FUNCTION_BLOCK FB_VirtualControlBox IMPLEMENTS I_ControlBox
VAR_INPUT
END_VAR
VAR_OUTPUT
END_VAR
VAR
END_VAR

//fbControlBox.Mode(
//	bAuto := VirtualControlBox.bAuto, 
//	bManual := VirtualControlBox.bManual,
//	eMode => VirtualControlBox.eMode
//);

//fbControlBox.Status(
//	eMode := VirtualControlBox.eMode,
//	bStart := VirtualControlBox.bSTART,
//	bStop := VirtualControlBox.bSTOP,
//	eStatus => VirtualControlBox.eStatus
//	);

{warning 'add method implementation '}
METHOD Joystick
VAR_INPUT
	//stJoystick	: ST_Joystick;
END_VAR
VAR_OUTPUT
	stJoystick : ST_Joystick;
END_VAR
VAR
	
END_VAR
ScaledInputs.stJoystick := VirtualControlBox.stJOY;

ScaledInputs.stJoystick.Topswitch := VirtualControlBox.stJOY.Topswitch;
//ScaledInputs.stJoystick := stJoystick;
END_METHOD

{warning 'add method implementation '}
METHOD Mode
VAR_INPUT
	//bAuto : BOOL;
	//bManual : BOOL;
	//eMode	: E_Mode; //should I read this value Directly from the VirtualControlBox?
END_VAR
VAR_OUTPUT
	eMode : E_Mode;
END_VAR

VAR
	//eMode : E_Mode;
	bAuto : BOOL;
	bManual : BOOL;
END_VAR
//eMode := VirtualControlBox.eMode;
//OUTPUTS.eMode := eMode;

bAuto := VirtualControlBox.bAuto;
bManual := VirtualControlBox.bManual;


IF bAuto AND NOT bManual THEN
	eMode := E_Mode.AUTO;
	Working.strMode := 'AUTO';
ELSIF bManual AND NOT bAuto THEN
	eMode := E_Mode.MANUAL;
	Working.strMode := 'MANUAL';
ELSE
	eMode := E_Mode.OFF;
	Working.strMode := 'OFF';
END_IF

Working.eMode := eMode;
END_METHOD

{warning 'add method implementation '}
METHOD Status
VAR_INPUT
	//eMode	: E_Mode;
	//bStart	: BOOL;
	//bStop	: BOOL;
END_VAR
VAR_OUTPUT
	//eStatus : E_Status := E_Status.NotReady;
END_VAR
VAR
	eStatus : E_Status;
	eMode : E_Mode;
END_VAR
eMode := Working.eMode;
eStatus := Working.eStatus;
CASE eStatus OF
	E_Status.NotReady:
		Working.strStatus := 'NotReady';
		IF eMode <> E_Mode.OFF THEN
			eStatus := E_Status.Ready;
		END_IF
	
	E_Status.Ready:
		Working.strStatus := 'Ready';
		IF eMode = E_Mode.OFF THEN
			eStatus := E_Status.NotReady;
		ELSIF VirtualControlBox.bStart THEN
			eStatus := E_Status.Starting;
		END_IF
		
	E_Status.Starting:
		Working.strStatus := 'Starting';
		IF VirtualControlBox.bStart AND NOT VirtualControlBox.bStop THEN //Add more start conditions?
			eStatus := E_Status.Running;	
		ELSE
			eStatus := E_Status.Ready;
		END_IF
		
	E_Status.Running:	
		Working.strStatus := 'Running';
		IF VirtualControlBox.bStop THEN
			eStatus := E_Status.Stopping;
		ELSIF eMode = E_Mode.AUTO THEN
			IF NOT VirtualControlBox.bStart THEN // ADD Clock signal
				eStatus := E_Status.Stopping;
			END_IF	
		END_IF
		
	E_Status.Stopping:
		Working.strStatus := 'Stopping';
		//Add stop condition
		eStatus := E_Status.NotReady;
		
	E_Status.Fault:
		Working.strStatus := 'Fault';				
END_CASE

Working.eStatus := eStatus;

////Control Lights
//IF eStatus = E_Status.Running THEN
//	OUTPUTS.bGreenLed := TRUE;
//	OUTPUTS.bEnableCylValve := TRUE;
//	IF ScaledInputs.stJoystick.Topswitch THEN
//		OUTPUTS.bEnableWinchValve := TRUE;
//	ELSE
//		OUTPUTS.bEnableWinchValve := FALSE;
//	END_IF
//ELSE
//	OUTPUTS.bGreenLed := FALSE;
//	OUTPUTS.bEnableCylValve := FALSE;
//	OUTPUTS.bEnableWinchValve := FALSE;
//END_IF

//IF eStatus = E_Status.Stopping OR eStatus = E_Status.Fault THEN
//	OUTPUTS.bRedLed := TRUE;
//ELSE
//	OUTPUTS.bRedLed := FALSE;
//END_IF
END_METHOD

END_FUNCTION_BLOCK

(* stored: Version 1.1.0.1, ProductVersion 3.1.4024.12
   POU FB_VirtualControlBox: Id {2aebf32b-d4cb-4b23-9b3a-2406c0f64e63}, SpecialFunc None
   Method Joystick: Id {5c488d52-6137-4781-8107-dc07e6a5f808}
   Method Mode: Id {2f785f0e-97f8-462b-9ade-1633aef6ec69}
   Method Status: Id {3a8a03aa-b9d0-43d2-ac17-130746f0a45c} *)
